{attribute addProperty BoxType "BK1150-0000-0016"}
{attribute addProperty Id "Term_383_KL1002KL1002_D229A9CA00"}
{attribute addProperty CRC "2132326926"}
{attribute addProperty SizeInBites "0"}
{attribute addProperty SizeInBytes "0"}
TYPE A_0010_BK1150_0000_0016_7F18BA0E EXTENDS BK1150_A5F67C82 :
STRUCT
	{attribute addProperty Name "Term_383_KL1002"}
	Term_383_KL1002 : KL1002_D229A9CA;
END_STRUCT
END_TYPE

(* stored: Version 1.2.0.0, ProductVersion 3.1.4024.9
   DUT A_0010_BK1150_0000_0016_7F18BA0E: Id {8692fd5d-f650-44a7-9e2d-03d2c28ad725} *)
